Staubli VAL3: onF2Event.pgx

program onF2Event(bool& x_bSave[])
  local string l_sEvent
  local num l_nIndex
  local num i
  local num l_nActualProg
  local string l_sMessage
  local string l_sButton[2]
  local bool l_bYes
  local string l_sResult
  local string l_sItem
  local string l_sEmpty
begin
  // look if the bButton is enable
  if bButton[1]
    // none
  endIf
end
